FUNCTION FC_BYTE_TO_BOOLBYTE : ARRAY[0..7] OF BOOL
VAR_INPUT
	myByte : REFERENCE TO BYTE;
END_VAR
VAR
    i : USINT;
END_VAR

FOR i := 0 TO 7 DO
    FC_BYTE_TO_BOOLBYTE[i] := (myByte AND (SHL(1,i))) <> 0;
END_FOR

END_FUNCTION

(* stored: Version 1.1.0.1, ProductVersion 3.1.4024.13
   POU FC_BYTE_TO_BOOLBYTE: Id {a8aa1d18-1612-476e-b910-0910d2267711}, SpecialFunc None *)
